Fanuc TP program (LS listing): BOTTOM01.LS

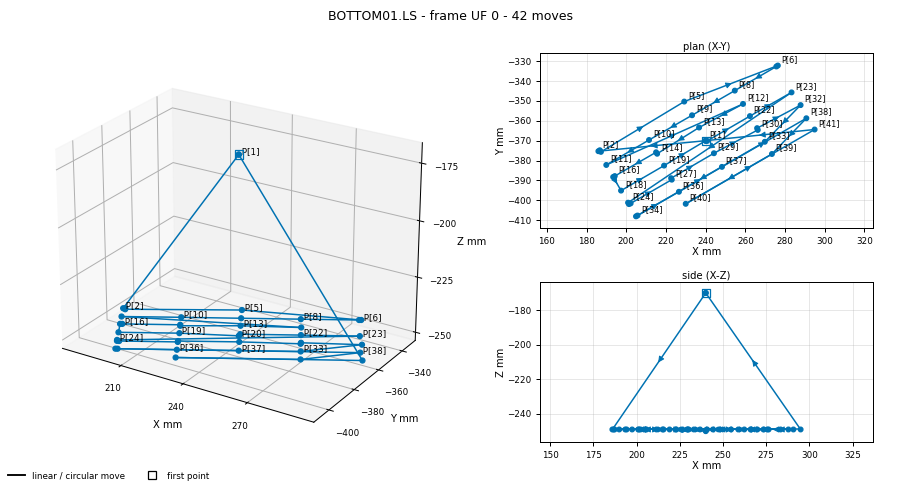
[picture p0: tool path of BOTTOM01.LS in frame UF 0, 42 of 42 moves have a stored position in this frame; points joined in program order, loops and branches not executed]
/PROG  BOTTOM01.LS
/ATTR
OWNER       = MNEDITOR;
COMMENT     = "";
PROG_SIZE   = 636;
CREATE      = DATE 23-01-07  TIME 11:59:14;
MODIFIED    = DATE 23-01-07  TIME 12:02:18;
FILE_NAME   = ;
VERSION     = 0;
LINE_COUNT  = 4;
MEMORY_SIZE = 992;
PROTECT     = READ_WRITE;
TCD:  STACK_SIZE	= 0,
      TASK_PRIORITY	= 50,
      TIME_SLICE	= 0,
      BUSY_LAMP_OFF	= 0,
      ABORT_REQUEST	= 0,
      PAUSE_REQUEST	= 0;
DEFAULT_GROUP	= 1,*,*,*,*;
CONTROL_CODE	= 00000000 00000000;
/MN
   1:J P[1] 100% FINE    ;
   2:L P[2] 100mm/sec CNT0    ;
   3:L P[3] 100mm/sec CNT0    ;
   4:L P[4] 100mm/sec CNT0    ;
   5:L P[5] 100mm/sec CNT0    ;
   6:L P[6] 100mm/sec CNT0    ;
   7:L P[7] 100mm/sec CNT0    ;
   8:L P[8] 100mm/sec CNT0    ;
   9:L P[9] 100mm/sec CNT0    ;
   10:L P[10] 100mm/sec CNT0    ;
   11:L P[11] 100mm/sec CNT0    ;
   12:L P[12] 100mm/sec CNT0    ;
   13:L P[13] 100mm/sec CNT0    ;
   14:L P[14] 100mm/sec CNT0    ;
   15:L P[15] 100mm/sec CNT0    ;
   16:L P[16] 100mm/sec CNT0    ;
   17:L P[17] 100mm/sec CNT0    ;
   18:L P[18] 100mm/sec CNT0    ;
   19:L P[19] 100mm/sec CNT0    ;
   20:L P[20] 100mm/sec CNT0    ;
   21:L P[21] 100mm/sec CNT0    ;
   22:L P[22] 100mm/sec CNT0    ;
   23:L P[23] 100mm/sec CNT0    ;
   24:L P[24] 100mm/sec CNT0    ;
   25:L P[25] 100mm/sec CNT0    ;
   26:L P[26] 100mm/sec CNT0    ;
   27:L P[27] 100mm/sec CNT0    ;
   28:L P[28] 100mm/sec CNT0    ;
   29:L P[29] 100mm/sec CNT0    ;
   30:L P[30] 100mm/sec CNT0    ;
   31:L P[31] 100mm/sec CNT0    ;
   32:L P[32] 100mm/sec CNT0    ;
   33:L P[33] 100mm/sec CNT0    ;
   34:L P[34] 100mm/sec CNT0    ;
   35:L P[35] 100mm/sec CNT0    ;
   36:L P[36] 100mm/sec CNT0    ;
   37:L P[37] 100mm/sec CNT0    ;
   38:L P[38] 100mm/sec CNT0    ;
   39:L P[39] 100mm/sec CNT0    ;
   40:L P[40] 100mm/sec CNT0    ;
   41:L P[41] 100mm/sec CNT0    ;
   42:L P[42] 100mm/sec CNT0    ;
/POS
P[1]{
   GP1:
	UF : 0, UT : 6,		CONFIG : 'N U T, 0, 0, 0',
	X =  240.000  mm,	Y =   -370.000  mm,	Z =   -170.000  mm,
	W =  90.000 deg,	P =   0.000 deg,	R =   30.000 deg
};
P[2]{
   GP1:
	UF : 0, UT : 6,		CONFIG : 'N U T, 0, 0, 0',
	X =  185.968  mm,	Y =   -375.301  mm,	Z =   -249.000  mm,
	W =  90.000 deg,	P =   0.000 deg,	R =   30.000 deg
};
P[3]{
   GP1:
	UF : 0, UT : 6,		CONFIG : 'N U T, 0, 0, 0',
	X =  186.708  mm,	Y =   -374.821  mm,	Z =   -249.000  mm,
	W =  90.000 deg,	P =   0.000 deg,	R =   30.000 deg
};
P[4]{
   GP1:
	UF : 0, UT : 6,		CONFIG : 'N U T, 0, 0, 0',
	X =  187.244  mm,	Y =   -375.631  mm,	Z =   -249.000  mm,
	W =  90.000 deg,	P =   0.000 deg,	R =   30.000 deg
};
P[5]{
   GP1:
	UF : 0, UT : 6,		CONFIG : 'N U T, 0, 0, 0',
	X =  229.225  mm,	Y =   -350.299  mm,	Z =   -249.000  mm,
	W =  90.000 deg,	P =   0.000 deg,	R =   30.000 deg
};
P[6]{
   GP1:
	UF : 0, UT : 6,		CONFIG : 'N U T, 0, 0, 0',
	X =  276.362  mm,	Y =   -332.143  mm,	Z =   -249.000  mm,
	W =  90.000 deg,	P =   0.000 deg,	R =   30.000 deg
};
P[7]{
   GP1:
	UF : 0, UT : 6,		CONFIG : 'N U T, 0, 0, 0',
	X =  275.617  mm,	Y =   -332.632  mm,	Z =   -249.000  mm,
	W =  90.000 deg,	P =   0.000 deg,	R =   30.000 deg
};
P[8]{
   GP1:
	UF : 0, UT : 6,		CONFIG : 'N U T, 0, 0, 0',
	X =  254.676  mm,	Y =   -344.782  mm,	Z =   -249.000  mm,
	W =  90.000 deg,	P =   0.000 deg,	R =   30.000 deg
};
P[9]{
   GP1:
	UF : 0, UT : 6,		CONFIG : 'N U T, 0, 0, 0',
	X =  233.148  mm,	Y =   -357.196  mm,	Z =   -249.000  mm,
	W =  90.000 deg,	P =   0.000 deg,	R =   30.000 deg
};
P[10]{
   GP1:
	UF : 0, UT : 6,		CONFIG : 'N U T, 0, 0, 0',
	X =  211.480  mm,	Y =   -369.654  mm,	Z =   -249.000  mm,
	W =  90.000 deg,	P =   0.000 deg,	R =   30.000 deg
};
P[11]{
   GP1:
	UF : 0, UT : 6,		CONFIG : 'N U T, 0, 0, 0',
	X =  189.944  mm,	Y =   -382.233  mm,	Z =   -249.000  mm,
	W =  90.000 deg,	P =   0.000 deg,	R =   30.000 deg
};
P[12]{
   GP1:
	UF : 0, UT : 6,		CONFIG : 'N U T, 0, 0, 0',
	X =  258.826  mm,	Y =   -351.488  mm,	Z =   -249.000  mm,
	W =  90.000 deg,	P =   0.000 deg,	R =   30.000 deg
};
P[13]{
   GP1:
	UF : 0, UT : 6,		CONFIG : 'N U T, 0, 0, 0',
	X =  236.702  mm,	Y =   -363.363  mm,	Z =   -249.000  mm,
	W =  90.000 deg,	P =   0.000 deg,	R =   30.000 deg
};
P[14]{
   GP1:
	UF : 0, UT : 6,		CONFIG : 'N U T, 0, 0, 0',
	X =  215.564  mm,	Y =   -376.583  mm,	Z =   -249.000  mm,
	W =  90.000 deg,	P =   0.000 deg,	R =   30.000 deg
};
P[15]{
   GP1:
	UF : 0, UT : 6,		CONFIG : 'N U T, 0, 0, 0',
	X =  215.032  mm,	Y =   -375.835  mm,	Z =   -249.000  mm,
	W =  90.000 deg,	P =   0.000 deg,	R =   30.000 deg
};
P[16]{
   GP1:
	UF : 0, UT : 6,		CONFIG : 'N U T, 0, 0, 0',
	X =  194.217  mm,	Y =   -387.839  mm,	Z =   -249.000  mm,
	W =  90.000 deg,	P =   0.000 deg,	R =   30.000 deg
};
P[17]{
   GP1:
	UF : 0, UT : 6,		CONFIG : 'N U T, 0, 0, 0',
	X =  193.424  mm,	Y =   -388.289  mm,	Z =   -249.000  mm,
	W =  90.000 deg,	P =   0.000 deg,	R =   30.000 deg
};
P[18]{
   GP1:
	UF : 0, UT : 6,		CONFIG : 'N U T, 0, 0, 0',
	X =  197.388  mm,	Y =   -395.153  mm,	Z =   -249.000  mm,
	W =  90.000 deg,	P =   0.000 deg,	R =   30.000 deg
};
P[19]{
   GP1:
	UF : 0, UT : 6,		CONFIG : 'N U T, 0, 0, 0',
	X =  219.058  mm,	Y =   -382.551  mm,	Z =   -249.000  mm,
	W =  90.000 deg,	P =   0.000 deg,	R =   30.000 deg
};
P[20]{
   GP1:
	UF : 0, UT : 6,		CONFIG : 'N U T, 0, 0, 0',
	X =  240.000  mm,	Y =   -370.000  mm,	Z =   -250.000  mm,
	W =  90.000 deg,	P =   0.000 deg,	R =   30.000 deg
};
P[21]{
   GP1:
	UF : 0, UT : 6,		CONFIG : 'N U T, 0, 0, 0',
	X =  240.755  mm,	Y =   -370.122  mm,	Z =   -249.000  mm,
	W =  90.000 deg,	P =   0.000 deg,	R =   30.000 deg
};
P[22]{
   GP1:
	UF : 0, UT : 6,		CONFIG : 'N U T, 0, 0, 0',
	X =  262.308  mm,	Y =   -357.619  mm,	Z =   -249.000  mm,
	W =  90.000 deg,	P =   0.000 deg,	R =   30.000 deg
};
P[23]{
   GP1:
	UF : 0, UT : 6,		CONFIG : 'N U T, 0, 0, 0',
	X =  283.264  mm,	Y =   -345.676  mm,	Z =   -249.000  mm,
	W =  90.000 deg,	P =   0.000 deg,	R =   30.000 deg
};
P[24]{
   GP1:
	UF : 0, UT : 6,		CONFIG : 'N U T, 0, 0, 0',
	X =  200.930  mm,	Y =   -401.229  mm,	Z =   -249.000  mm,
	W =  90.000 deg,	P =   0.000 deg,	R =   30.000 deg
};
P[25]{
   GP1:
	UF : 0, UT : 6,		CONFIG : 'N U T, 0, 0, 0',
	X =  201.372  mm,	Y =   -401.941  mm,	Z =   -249.000  mm,
	W =  90.000 deg,	P =   0.000 deg,	R =   30.000 deg
};
P[26]{
   GP1:
	UF : 0, UT : 6,		CONFIG : 'N U T, 0, 0, 0',
	X =  202.217  mm,	Y =   -401.593  mm,	Z =   -249.000  mm,
	W =  90.000 deg,	P =   0.000 deg,	R =   30.000 deg
};
P[27]{
   GP1:
	UF : 0, UT : 6,		CONFIG : 'N U T, 0, 0, 0',
	X =  222.935  mm,	Y =   -389.644  mm,	Z =   -249.000  mm,
	W =  90.000 deg,	P =   0.000 deg,	R =   30.000 deg
};
P[28]{
   GP1:
	UF : 0, UT : 6,		CONFIG : 'N U T, 0, 0, 0',
	X =  222.616  mm,	Y =   -388.901  mm,	Z =   -249.000  mm,
	W =  90.000 deg,	P =   0.000 deg,	R =   30.000 deg
};
P[29]{
   GP1:
	UF : 0, UT : 6,		CONFIG : 'N U T, 0, 0, 0',
	X =  244.172  mm,	Y =   -376.324  mm,	Z =   -249.000  mm,
	W =  90.000 deg,	P =   0.000 deg,	R =   30.000 deg
};
P[30]{
   GP1:
	UF : 0, UT : 6,		CONFIG : 'N U T, 0, 0, 0',
	X =  266.254  mm,	Y =   -364.590  mm,	Z =   -249.000  mm,
	W =  90.000 deg,	P =   0.000 deg,	R =   30.000 deg
};
P[31]{
   GP1:
	UF : 0, UT : 6,		CONFIG : 'N U T, 0, 0, 0',
	X =  265.930  mm,	Y =   -363.693  mm,	Z =   -249.000  mm,
	W =  90.000 deg,	P =   0.000 deg,	R =   30.000 deg
};
P[32]{
   GP1:
	UF : 0, UT : 6,		CONFIG : 'N U T, 0, 0, 0',
	X =  287.829  mm,	Y =   -352.076  mm,	Z =   -249.000  mm,
	W =  90.000 deg,	P =   0.000 deg,	R =   30.000 deg
};
P[33]{
   GP1:
	UF : 0, UT : 6,		CONFIG : 'N U T, 0, 0, 0',
	X =  269.812  mm,	Y =   -370.553  mm,	Z =   -249.000  mm,
	W =  90.000 deg,	P =   0.000 deg,	R =   30.000 deg
};
P[34]{
   GP1:
	UF : 0, UT : 6,		CONFIG : 'N U T, 0, 0, 0',
	X =  205.682  mm,	Y =   -407.704  mm,	Z =   -249.000  mm,
	W =  90.000 deg,	P =   0.000 deg,	R =   30.000 deg
};
P[35]{
   GP1:
	UF : 0, UT : 6,		CONFIG : 'N U T, 0, 0, 0',
	X =  204.922  mm,	Y =   -408.120  mm,	Z =   -249.000  mm,
	W =  90.000 deg,	P =   0.000 deg,	R =   30.000 deg
};
P[36]{
   GP1:
	UF : 0, UT : 6,		CONFIG : 'N U T, 0, 0, 0',
	X =  226.544  mm,	Y =   -395.739  mm,	Z =   -249.000  mm,
	W =  90.000 deg,	P =   0.000 deg,	R =   30.000 deg
};
P[37]{
   GP1:
	UF : 0, UT : 6,		CONFIG : 'N U T, 0, 0, 0',
	X =  248.211  mm,	Y =   -383.191  mm,	Z =   -249.000  mm,
	W =  90.000 deg,	P =   0.000 deg,	R =   30.000 deg
};
P[38]{
   GP1:
	UF : 0, UT : 6,		CONFIG : 'N U T, 0, 0, 0',
	X =  290.727  mm,	Y =   -358.709  mm,	Z =   -249.000  mm,
	W =  90.000 deg,	P =   0.000 deg,	R =   30.000 deg
};
P[39]{
   GP1:
	UF : 0, UT : 6,		CONFIG : 'N U T, 0, 0, 0',
	X =  273.382  mm,	Y =   -376.701  mm,	Z =   -249.000  mm,
	W =  90.000 deg,	P =   0.000 deg,	R =   30.000 deg
};
P[40]{
   GP1:
	UF : 0, UT : 6,		CONFIG : 'N U T, 0, 0, 0',
	X =  229.960  mm,	Y =   -401.807  mm,	Z =   -249.000  mm,
	W =  90.000 deg,	P =   0.000 deg,	R =   30.000 deg
};
P[41]{
   GP1:
	UF : 0, UT : 6,		CONFIG : 'N U T, 0, 0, 0',
	X =  294.889  mm,	Y =   -364.374  mm,	Z =   -249.000  mm,
	W =  90.000 deg,	P =   0.000 deg,	R =   30.000 deg
};
P[42]{
   GP1:
	UF : 0, UT : 6,		CONFIG : 'N U T, 0, 0, 0',
	X =  240.000  mm,	Y =   -370.000  mm,	Z =   -170.000  mm,
	W =  90.000 deg,	P =   0.000 deg,	R =   30.000 deg
};
/END
